Staubli VAL3: numCopy.pgx

public program numCopy(num& x_nCopy[] (dimensions=1), num& x_nPaste[] (dimensions=1))
// Copy all the value from the x_nCopy to x_nPaste
  local num i
  local num l_nSize
begin
  // Copy all the value from the first element to the second one
  //
  // redim the Paste String ARRAY
  //
  if size(x_nPaste)!=size(x_nCopy)
    resize(x_nPaste,1,size(x_nCopy))
  endIf
  // COPY ALL THE FIELD
  for i=0 to (size(x_nCopy)-1)
    x_nPaste[i]=x_nCopy[i]
  endFor
end
